// TwinCAT 3 PLC project OnGantryRTC_PLC
// ProgramVersion: 3.1.4020.4
// libraries:
//   Tc2_EtherCAT, * (Beckhoff Automation GmbH)
//   Tc2_Standard, * (Beckhoff Automation GmbH)
//   Tc2_System, * (Beckhoff Automation GmbH)
//   Tc3_Module, * (Beckhoff Automation GmbH)
// project tree:
//   / PlcTask.TcTTO
//   POUs/ BeamEnChain.TcPOU, bsm.TcPOU, Ehercat_Manage.TcPOU, F_scale_int_real.TcPOU, F_scale_real_int.TcPOU, OnGantry_IO.TcPOU
// real-time tasks:
//   TASK Task10ms: cycle T#10ms, priority 10, ADS port 350
//   TASK Task5ms: cycle T#5ms, priority 1, ADS port 351
//   TASK PlcTask: cycle T#10ms, priority 20, ADS port 352
// I/O:
//   DEVICE PCI, AmsNetId 192.168.60.2.2.1
//     Term 1 (EK1200) [EK1200-5000 EtherCAT Power supply (2A E-Bus)]
//       Term 2 (EL1809) [EL1809 16Ch. Dig. Input 24V, 3ms]
//       Term 3 (EL2809) [EL2809 16Ch. Dig. Output 24V, 0.5A]
//       Term 4 (EL6751) [EL6751 CANopen Master]
//       Term 5 (EL9011) [EL9011 End Terminal]
//   DEVICE MasterOut, AmsNetId 192.168.60.2.7.1
//     SlaveBSM [CX2030 EtherCAT slave]
//     SlaveBGM [CX2030 EtherCAT slave]
//     SlaveIGS [CX2030 EtherCAT slave]
//   DEVICE MasterIn (disabled), AmsNetId 192.168.60.2.4.1
//   DEVICE Device 5 (USB)
//     Box 1 (CX2100 Power Supply)
//     Box 254 (C9900-L100 License-Key-USB-Stick)
//   DEVICE CANOpenMaster, AmsNetId 192.168.60.2.3.1
//     Box 1 (EL6751)
//   DEVICE NRT
// variable links:
//   CANOpenMaster <-> RTC_StateMachine/ThreadFSM
//     Box 1 (EL6751)/Inputs/NodeState <-> FmDevices/CANOpen
//     Box 1 (EL6751)/RxPDO 1/Outputs/CurrentState <-> OutputsOGR/CurrentState
//     Box 1 (EL6751)/RxPDO 1/Outputs/DoseSegment <-> OutputsOGR/DoseSegment
//     Box 1 (EL6751)/RxPDO 1/Outputs/DoseTotal <-> OutputsOGR/DoseTotal
//     Box 1 (EL6751)/RxPDO 1/Outputs/IUT <-> OutputsOGR/IUT
//     Box 1 (EL6751)/RxPDO 2/Outputs/CollimatorDegree <-> OutputsBsm/CollimatorDegree
//     Box 1 (EL6751)/TxPDO 1/Inputs/CurrentState <-> InputsOGR/CurrentState
//     Box 1 (EL6751)/TxPDO 1/Inputs/GantryAngle <-> InputsOGR/GantryAngle
//     Box 1 (EL6751)/TxPDO 1/Inputs/GantrySpeed <-> InputsOGR/GantrySpeed
//     Box 1 (EL6751)/TxPDO 1/Inputs/IUT <-> InputsOGR/IUT
//     Box 1 (EL6751)/TxPDO 1/Inputs/RadiationIndex <-> InputsOGR/RadiationIndex
//     Box 1 (EL6751)/TxPDO 2/Inputs/FieldDefiningLamp <-> InputsBsm/FieldLightFrmBSC
//     Box 1 (EL6751)/TxPDO 2/Inputs/FkpButton <-> InputsOGR/FkpButton
//     Box 1 (EL6751)/TxPDO 2/Inputs/OdiLight <-> InputsBsm/OdiLight
//     Box 1 (EL6751)/TxPDO 3/Inputs/BsmMotionEnable <-> InputsBsm/BsmMotionEnable
//     Box 1 (EL6751)/TxPDO 3/Inputs/HHCWheel1 <-> InputsBsm/WheelBsm1
//     Box 1 (EL6751)/TxPDO 3/Inputs/HHCWheel2 <-> InputsBsm/WheelBsm2
//     Box 1 (EL6751)/TxPDO 3/Inputs/HHCWheel3 <-> InputsBsm/WheelBsm3
//   MasterOut <-> RTC_StateMachine/ThreadFSM
//     SlaveBGM/IO Inputs/BankIndex <-> InputsBgmPlan/BankIndex
//     SlaveBGM/IO Inputs/BeamID <-> InputsBgmPlan/BeamID
//     SlaveBGM/IO Inputs/CPIndex <-> InputsBgmPlan/CPIndex
//     SlaveBGM/IO Inputs/CPTotal <-> InputsBgmPlan/CPTotal
//     SlaveBGM/IO Inputs/Crc32 <-> InputsBgmPlan/Crc32
//     SlaveBGM/IO Inputs/DoseSegment <-> InputsDose/DoseSegment
//     SlaveBGM/IO Inputs/DoseTotal <-> InputsDose/DoseTotal
//     SlaveBGM/IO Inputs/RadiationIndex <-> InputsBeam/RadiationIndex
//     SlaveBGM/IO Inputs/WatchDogOk <-> FmDevices/BgmWdOk
//     SlaveBGM/IO Inputs/bgm_interlocks <-> InputsSubFsm/BgmInterlocks
//     SlaveBGM/IO Inputs/bgm_last_state <-> InputsSubFsm/BgmLastState
//     SlaveBGM/IO Inputs/bgm_required_state <-> InputsSubFsm/BgmRequiredState
//     SlaveBGM/IO Inputs/bgm_state <-> InputsSubFsm/BgmCurrentState
//     SlaveBGM/IO Inputs/bgm_unready1 <-> InputsSubFsm/BgmUnreadys
//     SlaveBGM/IO Outputs/BankIndex <-> OutputsBgmPlan/BankIndex
//     SlaveBGM/IO Outputs/BeamID <-> OutputsBgmPlan/BeamID
//     SlaveBGM/IO Outputs/CPIndex <-> OutputsBgmPlan/CPIndex
//     SlaveBGM/IO Outputs/CPTotal <-> OutputsBgmPlan/CPTotal
//     SlaveBGM/IO Outputs/Crc32 <-> OutputsBgmPlan/Crc32
//     SlaveBGM/IO Outputs/DoseInterlockEnable <-> OutputsDose/DoseInterlockEnable
//     SlaveBGM/IO Outputs/DoseTotal <-> OutputsBgmPlan/DoseTotal
//     SlaveBGM/IO Outputs/PlanData <-> OutputsBgmPlan/Data
//     SlaveBGM/IO Outputs/QuickBeamTotalSet1 <-> OutputsBeam/beam_total_set1
//     SlaveBGM/IO Outputs/RadiationIndex <-> OutputsOGR/RadiationIndex
//     SlaveBGM/IO Outputs/RequiredState <-> OutputsSubFsm/BgmRequiredState
//     SlaveBGM/IO Outputs/ServoAxisType <-> OutputsBgmPlan/ServoAxisType
//     SlaveBGM/InfoData/State <-> FmDevices/BGMSlave
//     SlaveBSM/IO Inputs/BankIndex <-> InputsBsm/BankIndex
//     SlaveBSM/IO Inputs/BeamId <-> InputsBsm/BeamID
//     SlaveBSM/IO Inputs/BsmReady <-> InputsBsm/BsmReady
//     SlaveBSM/IO Inputs/CollimatorPosition <-> InputsBsm/CollimatorPosition
//     SlaveBSM/IO Inputs/CpIndex <-> InputsBsm/CPIndex
//     SlaveBSM/IO Inputs/CpTotal <-> InputsBsm/CPTotal
//     SlaveBSM/IO Inputs/Crc32 <-> InputsBsm/Crc32
//     SlaveBSM/IO Inputs/CurrentState <-> InputsBsm/CurrentState
//     SlaveBSM/IO Inputs/Data <-> InputsBsm/PosFeedback
//     SlaveBSM/IO Inputs/HeadP1 <-> InputsBsm/HeadP1
//     SlaveBSM/IO Inputs/HeaddSpeed <-> InputsBsm/HeadSpeed
//     SlaveBSM/IO Inputs/Headp2 <-> InputsBsm/HeadP2
//     SlaveBSM/IO Inputs/InitModeAck <-> InputsBsm/BSMInitModeAck
//     SlaveBSM/IO Inputs/InitResult1 <-> InputsBsm/InitResult1
//     SlaveBSM/IO Inputs/InitResult2 <-> InputsBsm/InitResult2
//     SlaveBSM/IO Inputs/Interlock <-> InputsBsm/Interlock
//     SlaveBSM/IO Inputs/JawMaxSpeed <-> InputsBsm/JawMaxSpeed
//     SlaveBSM/IO Inputs/LastState <-> InputsBsm/LastState
//     SlaveBSM/IO Inputs/LeafMaxSpeed <-> InputsBsm/LeafMaxSpeed
//     SlaveBSM/IO Inputs/RadiationIndex <-> InputsBsm/RadiationIndex
//     SlaveBSM/IO Inputs/Status <-> InputsBsm/Status
//     SlaveBSM/IO Inputs/UpJaw1P1 <-> InputsBsm/UpJaw1P1
//     SlaveBSM/IO Inputs/UpJaw1P2 <-> InputsBsm/UpJaw1P2
//     SlaveBSM/IO Inputs/UpJaw2P1 <-> InputsBsm/UpJaw2P1
//     SlaveBSM/IO Inputs/UpJaw2P2 <-> InputsBsm/UpJaw2P2
//     SlaveBSM/IO Outputs/BSMInitMode <-> OutputsBsm/BSMInitMode
//     SlaveBSM/IO Outputs/BSMOK <-> OutputsBsm/BsmOk
//     SlaveBSM/IO Outputs/BankIndex <-> OutputsBsm/BankIndex
//     SlaveBSM/IO Outputs/BeamId <-> OutputsBsm/BeamID
//     SlaveBSM/IO Outputs/CalibrationJaw <-> OutputsBsm/CalibrationJaw
//     SlaveBSM/IO Outputs/CollimatorPosition <-> OutputsBsm/CollimatorPosition
//     SlaveBSM/IO Outputs/Commands <-> OutputsBsm/Commands
//     SlaveBSM/IO Outputs/CpIndex <-> OutputsBsm/CPIndex
//     SlaveBSM/IO Outputs/CpTotal <-> OutputsBsm/CPTotal
//     SlaveBSM/IO Outputs/Crc32 <-> OutputsBsm/Crc32
//     SlaveBSM/IO Outputs/Data <-> OutputsBsm/Data
//     SlaveBSM/IO Outputs/HHCFunctionCode <-> OutputsBsm/HhcFunctionCode
//     SlaveBSM/IO Outputs/HHCVoltage <-> OutputsBsm/HhcVoltage
//     SlaveBSM/IO Outputs/HHCWheel1 <-> OutputsBsm/HHCWheel1
//     SlaveBSM/IO Outputs/HHCWheel2 <-> OutputsBsm/HHCWheel2
//     SlaveBSM/IO Outputs/HHCWheel3 <-> OutputsBsm/HHCWheel3
//     SlaveBSM/IO Outputs/HeadAngle <-> OutputsBsm/HeadAngle
//     SlaveBSM/IO Outputs/HeadAngleK <-> OutputsBsm/HeadAngleK
//     SlaveBSM/IO Outputs/HeadAngleOffset <-> OutputsBsm/HeadAngleOffset
//     SlaveBSM/IO Outputs/HeadAngleSecondaryK <-> OutputsBsm/HeadAngleSecondaryK
//     SlaveBSM/IO Outputs/HeadLimitEncoder <-> OutputsBsm/HeadLimitEncoder
//     SlaveBSM/IO Outputs/HeadSpeed <-> OutputsBsm/HeadSpeed
//     SlaveBSM/IO Outputs/HeadTolerance <-> OutputsBsm/HeadTolerance
//     SlaveBSM/IO Outputs/HwEnable <-> OutputsBsm/HwEnable
//     SlaveBSM/IO Outputs/JawXTolerance <-> OutputsBsm/ToleranceJawX
//     SlaveBSM/IO Outputs/JawYTolerance <-> OutputsBsm/ToleranceJawY
//     SlaveBSM/IO Outputs/LeafTolerance <-> OutputsBsm/ToleranceLeaf
//     SlaveBSM/IO Outputs/RadiationIndex <-> OutputsBsm/RadiationIndex
//     SlaveBSM/IO Outputs/RequiredState <-> OutputsBsm/RequiredState
//     SlaveBSM/IO Outputs/UpJaw1Pos <-> OutputsBsm/UpJaw1Pos
//     SlaveBSM/IO Outputs/UpJaw2Pos <-> OutputsBsm/UpJaw2Pos
//     SlaveBSM/IO Outputs/UpJaw1Speed <-> OutputsBsm/UpJaw1Speed
//     SlaveBSM/IO Outputs/UpJaw2Speed <-> OutputsBsm/UpJaw2Speed
//     SlaveBSM/InfoData/State <-> FmDevices/BSMSlave
//     SlaveIGS/IO Inputs/CollimatorCross <-> InputsIgsSlv/CollimatorCross
//     SlaveIGS/IO Inputs/CollimatorLong <-> InputsIgsSlv/CollimatorLong
//     SlaveIGS/IO Inputs/CollimatorOffsetCross <-> InputsIgsSlv/CollimatorOffsetCross
//     SlaveIGS/IO Inputs/CollimatorOffsetLong <-> InputsIgsSlv/CollimatorOffsetLong
//     SlaveIGS/IO Inputs/CollimatorPosReady <-> InputsIgsSlv/CollimatorPosReady
//     SlaveIGS/IO Inputs/CurrentState <-> InputsIgsSlv/CurrentState
//     SlaveIGS/IO Inputs/HighVoltageGeneratorErrorCode <-> InputsIgsSlv/HighVoltageGeneratorErrorCode
//     SlaveIGS/IO Inputs/ICUFocusExpActual <-> InputsIgsSlv/IcuFocusExpActual
//     SlaveIGS/IO Inputs/ICUFrequencyExpActual <-> InputsIgsSlv/IcuFrequencyExpActual
//     SlaveIGS/IO Inputs/ICUKVExpActual <-> InputsIgsSlv/IcuKVExpActual
//     SlaveIGS/IO Inputs/ICUMAExpActual <-> InputsIgsSlv/IcuMAExpActual
//     SlaveIGS/IO Inputs/ICUMSExpActual <-> InputsIgsSlv/IcuMSExpActual
//     SlaveIGS/IO Inputs/IcuErrorCode <-> InputsIgsSlv/IcuErrorCode
//     SlaveIGS/IO Inputs/Interlock <-> InputsIgsSlv/Interlock
//     SlaveIGS/IO Inputs/KVEncode1 <-> InputsIgsSlv/KVEncode1
//     SlaveIGS/IO Inputs/KVEncode2 <-> InputsIgsSlv/KVEncode2
//     SlaveIGS/IO Inputs/KVPosActual <-> InputsIgsSlv/KVPosActual
//     SlaveIGS/IO Inputs/KVPosReady <-> InputsIgsSlv/KVPosReady
//     SlaveIGS/IO Inputs/KvPanelErrorcode <-> InputsIgsSlv/KvPanelErrorcode
//     SlaveIGS/IO Inputs/LastState <-> InputsIgsSlv/LastState
//     SlaveIGS/IO Inputs/MVEncode1 <-> InputsIgsSlv/MVEncode1
//     SlaveIGS/IO Inputs/MVEncode2 <-> InputsIgsSlv/MVEncode2
//     SlaveIGS/IO Inputs/MVPanelErrorcode <-> InputsIgsSlv/MVPanelErrorcode
//     SlaveIGS/IO Inputs/MVPosActual <-> InputsIgsSlv/MVPosActual
//     SlaveIGS/IO Inputs/MVPosReady <-> InputsIgsSlv/MVPosReady
//     SlaveIGS/IO Inputs/RecordCounter <-> InputsIgsSlv/RecordCounter
//     SlaveIGS/IO Inputs/RecordFlag <-> InputsIgsSlv/RecordFlag
//     SlaveIGS/IO Inputs/WatchDogOk <-> FmDevices/IgsWdOk
//     SlaveIGS/IO Outputs/CollimatorCross <-> OutputsIgsSlv/CollimatorCross
//     SlaveIGS/IO Outputs/CollimatorLong <-> OutputsIgsSlv/CollimatorLong
//     SlaveIGS/IO Outputs/CollimatorOffsetCross <-> OutputsIgsSlv/CollimatorOffsetCross
//     SlaveIGS/IO Outputs/CollimatorOffsetLong <-> OutputsIgsSlv/CollimatorOffsetLong
//     SlaveIGS/IO Outputs/ICUFocusExp <-> OutputsIgsSlv/IcuFocusExp
//     SlaveIGS/IO Outputs/ICUFrequencyExp <-> OutputsIgsSlv/IcuFrequencyExp
//     SlaveIGS/IO Outputs/ICUKVExp <-> OutputsIgsSlv/IcuKVExp
//     SlaveIGS/IO Outputs/ICUMAExp <-> OutputsIgsSlv/IcuMAExp
//     SlaveIGS/IO Outputs/ICUMSExp <-> OutputsIgsSlv/IcuMSExp
//     SlaveIGS/IO Outputs/KVOffset1 <-> OutputsIgsSlv/KVOffset1
//     SlaveIGS/IO Outputs/KVOffset2 <-> OutputsIgsSlv/KVOffset2
//     SlaveIGS/IO Outputs/KVPosTarget <-> OutputsIgsSlv/KVPosTarget
//     SlaveIGS/IO Outputs/KvTimeout <-> OutputsIgsSlv/KvTimeout
//     SlaveIGS/IO Outputs/MVOffset1 <-> OutputsIgsSlv/MVOffset1
//     SlaveIGS/IO Outputs/MVOffset2 <-> OutputsIgsSlv/MVOffset2
//     SlaveIGS/IO Outputs/MVPosTarget <-> OutputsIgsSlv/MVPosTarget
//     SlaveIGS/IO Outputs/MvTimeout <-> OutputsIgsSlv/MvTimeout
//     SlaveIGS/IO Outputs/PlanTotalFrame <-> OutputsIgsSlv/PlanTotalFrame
//     SlaveIGS/IO Outputs/RequiredState <-> OutputsIgsSlv/RequiredState
//     SlaveIGS/IO Outputs/Reset <-> OutputsIgsSlv/Reset
//     SlaveIGS/IO Outputs/WorkMode <-> OutputsIgsSlv/WorkMode
//     SlaveIGS/InfoData/State <-> FmDevices/IGSSlave
//   MasterOut <-> TCPServer/ThreadGUI
//     SlaveBGM/IO Inputs/BgmHalEmulate <-> InputsHalState/EmulateState/BGM
//     SlaveBGM/IO Inputs/DoseDelta <-> InputsBeam/DoseDelta
//     SlaveBGM/IO Inputs/DoseInformation1 <-> InputsDose/DoseInformation1
//     SlaveBGM/IO Inputs/DoseInformation2 <-> InputsDose/DoseInformation2
//     SlaveBGM/IO Inputs/GunCathodCurrentRead <-> InputsGun/gun_cathode_current_read
//     SlaveBGM/IO Inputs/GunFilaCurrentRead <-> InputsGun/gun_fila_current_read
//     SlaveBGM/IO Inputs/GunFilaVolRead <-> InputsGun/gun_fila_vol_read
//     SlaveBGM/IO Inputs/GunHvRead <-> InputsGun/gun_hv_read
//     SlaveBGM/IO Inputs/GunRemainingTime <-> InputsGun/GunRemainingTime
//     SlaveBGM/IO Inputs/afc_RF_AI <-> InputsAfc/afc_RF_AI
//     SlaveBGM/IO Inputs/afc_current_pos <-> InputsAfc/afc_current_pos
//     SlaveBGM/IO Inputs/afc_mode <-> InputsAfc/afc_mode
//     SlaveBGM/IO Inputs/beam_dose_rate_read1 <-> InputsBeam/beam_dose_rate_read1
//     SlaveBGM/IO Inputs/beam_dose_rate_read2 <-> InputsBeam/beam_dose_rate_read2
//     SlaveBGM/IO Inputs/beam_total_read1 <-> InputsBeam/beam_total_read1
//     SlaveBGM/IO Inputs/beam_total_read2 <-> InputsBeam/beam_total_read2
//     SlaveBGM/IO Inputs/mod_app_ver <-> InputsModulator/mod_app_ver
//     SlaveBGM/IO Inputs/mod_average_power_read <-> InputsModulator/mod_average_power_read
//     SlaveBGM/IO Inputs/mod_dc_vol_read <-> InputsModulator/mod_dc_vol_read
//     SlaveBGM/IO Inputs/mod_dc_voltage_rb <-> InputsModulator/mod_dc_voltage_set_read
//     SlaveBGM/IO Inputs/mod_filament_current_read <-> InputsModulator/mod_filament_current_read
//     SlaveBGM/IO Inputs/mod_filament_vol_rb <-> InputsModulator/mod_filament_vol_set_read
//     SlaveBGM/IO Inputs/mod_filament_vol_read <-> InputsModulator/mod_filament_vol_read
//     SlaveBGM/IO Inputs/mod_fpga_ver <-> InputsModulator/mod_fpga_ver
//     SlaveBGM/IO Inputs/mod_hv_hour <-> InputsModulator/mod_hv_hour
//     SlaveBGM/IO Inputs/mod_hv_interlock <-> InputsModulator/mod_hv_interlock
//     SlaveBGM/IO Inputs/mod_level <-> InputsModulator/mod_level
//     SlaveBGM/IO Inputs/mod_off_hour <-> InputsModulator/mod_off_hour
//     SlaveBGM/IO Inputs/mod_pluse_width_rb <-> InputsModulator/mod_pulse_width_set_read
//     SlaveBGM/IO Inputs/mod_prf_read <-> InputsModulator/mod_prf_read
//     SlaveBGM/IO Inputs/mod_pulse_width_read <-> InputsModulator/mod_pulse_width_read
//     SlaveBGM/IO Inputs/mod_remaining_time <-> InputsModulator/mod_remaining_time
//     SlaveBGM/IO Inputs/mod_standby_hour <-> InputsModulator/mod_standby_hour
//     SlaveBGM/IO Inputs/mod_standby_interlock <-> InputsModulator/mod_standby_interlock
//     SlaveBGM/IO Inputs/mod_state_rb <-> InputsModulator/mod_state_set_read
//     SlaveBGM/IO Inputs/mod_state_read <-> InputsModulator/mod_state_read
//     SlaveBGM/IO Inputs/mod_trig_hour <-> InputsModulator/mod_trig_hour
//     SlaveBGM/IO Inputs/mod_trig_interlock <-> InputsModulator/mod_trig_interlock
//     SlaveBGM/IO Inputs/sf6_pressure <-> InputsSF6/sf6_pressure
//     SlaveBGM/IO Inputs/vac_current <-> InputsVac/vac_current
//     SlaveBGM/IO Inputs/vac_voltage <-> InputsVac/vac_voltage
//     SlaveBGM/IO Inputs/water_flow_in <-> InputsWater/water_flow_in
//     SlaveBGM/IO Inputs/water_flow_low_set <-> InputsWater/water_flow_low_set
//     SlaveBGM/IO Inputs/water_flow_switch <-> InputsWater/water_flow_switch
//     SlaveBGM/IO Inputs/water_interlock_raw <-> InputsWater/water_interlock_raw
//     SlaveBGM/IO Inputs/water_pressure_in <-> InputsWater/water_pressure
//     SlaveBGM/IO Inputs/water_temp_{1..5} <-> InputsWater/water_temp_{1..5}  (5 links)
//     SlaveBGM/IO Inputs/water_temp_back <-> InputsWater/water_temp_back
//     SlaveBGM/IO Inputs/water_temp_high_set <-> InputsWater/water_temp_high_set
//     SlaveBGM/IO Inputs/water_temp_in <-> InputsWater/water_temp_in
//     SlaveBGM/IO Inputs/water_temp_low_set <-> InputsWater/water_temp_low_set
//     SlaveBGM/IO Outputs/AfcRfSet <-> OutputsAfc/afc_RF_set
//     SlaveBGM/IO Outputs/DPP <-> OutputsPrf/DPP
//     SlaveBGM/IO Outputs/DarkCurrentLimit <-> OutputsDose/DarkCurrentLimit
//     SlaveBGM/IO Outputs/DoseCalFactorA1 <-> OutputsDose/DoseCalFactorA1
//     SlaveBGM/IO Outputs/DoseCalFactorA2 <-> OutputsDose/DoseCalFactorA2
//     SlaveBGM/IO Outputs/DoseCalFactorB1 <-> OutputsDose/DoseCalFactorB1
//     SlaveBGM/IO Outputs/DoseCalFactorB2 <-> OutputsDose/DoseCalFactorB2
//     SlaveBGM/IO Outputs/DoseDeltaActionRange <-> OutputsPrf/DoseDeltaActionRange
//     SlaveBGM/IO Outputs/DoseOverrangeRatio <-> OutputsDose/SegmentOverrangeRatio
//     SlaveBGM/IO Outputs/DoseRateAccTime <-> OutputsDose/DoseRateAccTime
//     SlaveBGM/IO Outputs/DoseRateCycleTime <-> OutputsDose/DoseRateCycleTime
//     SlaveBGM/IO Outputs/DoseRateLimit <-> OutputsDose/DoseRateLimit
//     SlaveBGM/IO Outputs/DualChannelRatio <-> OutputsDose/DualChannelRatio
//     SlaveBGM/IO Outputs/DualChannelTolerance <-> OutputsDose/DualChannelTolerance
//     SlaveBGM/IO Outputs/DummyDoseRateSet <-> OutputsDose/DummyDoseRateSet
//     SlaveBGM/IO Outputs/PrfCatchCurveD1 <-> OutputsPrf/PrfCatchCurveD1
//     SlaveBGM/IO Outputs/PrfCatchCurveD2 <-> OutputsPrf/PrfCatchCurveD2
//     SlaveBGM/IO Outputs/PrfCatchCurveP1 <-> OutputsPrf/PrfCatchCurveP1
//     SlaveBGM/IO Outputs/PrfCatchCurveP2 <-> OutputsPrf/PrfCatchCurveP2
//     SlaveBGM/IO Outputs/PrfCatchCurveQ1 <-> OutputsPrf/PrfCatchCurveQ1
//     SlaveBGM/IO Outputs/PrfCatchCurveQ2 <-> OutputsPrf/PrfCatchCurveQ2
//     SlaveBGM/IO Outputs/PrfCatchCurveR1 <-> OutputsPrf/PrfCatchCurveR1
//     SlaveBGM/IO Outputs/PrfCatchCurveR2 <-> OutputsPrf/PrfCatchCurveR2
//     SlaveBGM/IO Outputs/PrfCatchCycle <-> OutputsPrf/PrfCatchCycle
//     SlaveBGM/IO Outputs/PrfDeltaRatio <-> OutputsPrf/PrfDeltaRatio
//     SlaveBGM/IO Outputs/PrfRatio <-> OutputsPrf/PrfRatio
//     SlaveBGM/IO Outputs/QuickBeamProtectTimeSet <-> OutputsBeam/beam_time_set
//     SlaveBGM/IO Outputs/QuickBeamTotalSet2 <-> OutputsBeam/beam_total_set2
//     SlaveBGM/IO Outputs/SymmetryThreshold1 <-> OutputsDose/SymmetryThreshold1
//     SlaveBGM/IO Outputs/SymmetryThreshold2 <-> OutputsDose/SymmetryThreshold2
//     SlaveBGM/IO Outputs/SymmetryTolerance1 <-> OutputsDose/SymmetryTolerance1
//     SlaveBGM/IO Outputs/SymmetryTolerance2 <-> OutputsDose/SymmetryTolerance2
//     SlaveBGM/IO Outputs/afc_dir_swap <-> OutputsAfc/afc_dir_swap
//     SlaveBGM/IO Outputs/afc_linear_high <-> OutputsAfc/afc_linear_high
//     SlaveBGM/IO Outputs/afc_linear_low <-> OutputsAfc/afc_linear_low
//     SlaveBGM/IO Outputs/afc_manual_dir <-> OutputsAfc/afc_manual_dir
//     SlaveBGM/IO Outputs/afc_manual_move <-> OutputsAfc/afc_manual_move
//     SlaveBGM/IO Outputs/afc_mode_set <-> OutputsAfc/afc_mode_set
//     SlaveBGM/IO Outputs/afc_motor_max_speed <-> OutputsAfc/afc_motor_max_speed
//     SlaveBGM/IO Outputs/afc_preset <-> OutputsAfc/afc_preset
//     SlaveBGM/IO Outputs/emulator_enable <-> OutputsHalState/BgmEmulate
//     SlaveBGM/IO Outputs/gui_cmd_reset <-> OutputsFsm/reset_command
//     SlaveBGM/IO Outputs/gun_cathode_current_max <-> OutputsGun/gun_cathode_current_max
//     SlaveBGM/IO Outputs/gun_cathode_current_min <-> OutputsGun/gun_cathode_current_min
//     SlaveBGM/IO Outputs/gun_cathode_current_rat_2 <-> OutputsGun/gun_cathode_current_rat_2
//     SlaveBGM/IO Outputs/gun_dr_at_fullpower <-> OutputsGun/gun_dr_at_fullpower
//     SlaveBGM/IO Outputs/gun_fila_current_rat_2 <-> OutputsGun/gun_fila_current_rat_2
//     SlaveBGM/IO Outputs/gun_fila_current_set_tol <-> OutputsGun/gun_fila_current_set_tol
//     SlaveBGM/IO Outputs/gun_fila_vol_max <-> OutputsGun/gun_fila_vol_max
//     SlaveBGM/IO Outputs/gun_fila_vol_min <-> OutputsGun/gun_fila_vol_min
//     SlaveBGM/IO Outputs/gun_fila_vol_rat_2 <-> OutputsGun/gun_fila_vol_rat_2
//     SlaveBGM/IO Outputs/gun_fila_vol_set_rat_{1..4} <-> OutputsGun/gun_fila_vol_set_rat_{1..4}  (4 links)
//     SlaveBGM/IO Outputs/gun_heaterok_judgetime <-> OutputsGun/gun_heaterok_judgetime
//     SlaveBGM/IO Outputs/gun_hv <-> OutputsGun/gun_hv
//     SlaveBGM/IO Outputs/gun_hv_rat_{1..4} <-> OutputsGun/gun_hv_rat_{1..4}  (4 links)
//     SlaveBGM/IO Outputs/gun_hv_read_rat2 <-> OutputsGun/gun_hv_read_rat2
//     SlaveBGM/IO Outputs/gun_rundown_dr_k <-> OutputsGun/gun_rundown_dr_k
//     SlaveBGM/IO Outputs/gun_rundown_prf_k <-> OutputsGun/gun_rundown_prf_k
//     SlaveBGM/IO Outputs/gun_warmup <-> OutputsGun/gun_warmup
//     SlaveBGM/IO Outputs/gun_warmup_time <-> OutputsGun/gun_warmup_time
//     SlaveBGM/IO Outputs/mod_dc_voltage <-> OutputsModulator/mod_dc_voltage
//     SlaveBGM/IO Outputs/mod_filament_vol <-> OutputsModulator/mod_filament_vol
//     SlaveBGM/IO Outputs/mod_pulse_width <-> OutputsModulator/mod_pluse_width
//     SlaveBGM/IO Outputs/prf_set <-> OutputsPrf/prf_set
//     SlaveIGS/IO Inputs/HVGeneratorHU <-> InputsIgs/HVGeneratorHU
//     SlaveIGS/IO Outputs/KvTorlerance <-> OutputsIgs/KvTorlerance
//     SlaveIGS/IO Outputs/MvTorlerance <-> OutputsIgs/MvTorlerance
//   OnGantryRTC_PLC/OnGantryRTC_PLC Instance <-> MasterOut
//     PlcTask Inputs/Ehercat_Manage.arrbyNetId <-> InfoData/AmsNetId
//   OnGantryRTC_PLC/OnGantryRTC_PLC Instance <-> PCI/Term 1 (EK1200)/Term 2 (EL1809)
//     PlcTask Inputs/OnGantry_IO.plc_to_io_OnGantryRtcWdOK <-> Channel 3/Input
//     PlcTask Inputs/OnGantry_IO.plc_to_io_bAutoMove <-> Channel 2/Input
//     PlcTask Inputs/OnGantry_IO.plc_to_io_bGantryTouchGuard <-> Channel 1/Input
//   OnGantryRTC_PLC/OnGantryRTC_PLC Instance <-> PCI/Term 1 (EK1200)/Term 3 (EL2809)
//     PlcTask Outputs/OnGantry_IO.plc_to_io_OnGantryMoveEn <-> Channel 3/Output
//     PlcTask Outputs/OnGantry_IO.plc_to_io_bCanOpenOk <-> Channel 1/Output
//     PlcTask Outputs/OnGantry_IO.plc_to_io_bEthercatInOk <-> Channel 2/Output
//     PlcTask Outputs/OnGantry_IO.plc_to_io_bEthercatOutOk <-> Channel 4/Output
//     PlcTask Outputs/OnGantry_IO.plc_to_io_bKvEn <-> Channel 7/Output
//     PlcTask Outputs/OnGantry_IO.plc_to_io_bSwManualMotionEn <-> Channel 9/Output
//     PlcTask Outputs/OnGantry_IO.plc_to_io_bSwRest <-> Channel 6/Output
//     PlcTask Outputs/OnGantry_IO.plc_to_io_bSwWatchDogService <-> Channel 5/Output
//   OnGantryRTC_PLC/OnGantryRTC_PLC Instance <-> RTC_StateMachine/ThreadFSM
//     PlcTask Inputs/OnGantry_IO.plc_to_cpp_OnGantryMoveEn <-> OutputsOnGantryHD/SwOnGantryMoveEn
//     PlcTask Inputs/OnGantry_IO.plc_to_cpp_bCanOpenOk <-> OutputsOnGantryHD/SwCanOpenOk
//     PlcTask Inputs/OnGantry_IO.plc_to_cpp_bEthercatInOk <-> OutputsOnGantryHD/SwEthercatInOk
//     PlcTask Inputs/OnGantry_IO.plc_to_cpp_bEthercatOutOk <-> OutputsOnGantryHD/SwEthercatOutOk
//     PlcTask Inputs/OnGantry_IO.plc_to_cpp_bKvEn <-> OutputsOnGantryHD/SwKvEn
//     PlcTask Inputs/OnGantry_IO.plc_to_cpp_bSwManualMotionEn <-> OutputsFsm/bSwManualMotionEn
//     PlcTask Outputs/OnGantry_IO.plc_to_cpp_OnGantryRtcWdOK <-> FmDevices/OnGantryRTCWdOk
//     PlcTask Outputs/OnGantry_IO.plc_to_cpp_bAutoMove <-> InputsOnGantryHD/AutoMoveEn
//     PlcTask Outputs/OnGantry_IO.plc_to_cpp_bGantryTouchGuard <-> InputsOnGantryHD/GantryTouchGuard
//   OnGantryRTC_PLC/OnGantryRTC_PLC Instance <-> TCPServer/ThreadGUI
//     PlcTask Inputs/Ehercat_Manage.bResetState <-> OutputsFsm/reset_command
//     PlcTask Inputs/OnGantry_IO.plc_to_cpp_bSwRest <-> OutputsFsm/reset_command
//   RTC_StateMachine/ThreadFSM <-> TCPServer/ThreadGUI
//     InputsBeam/DoseRateSet <-> OutputsBeam/beam_dose_rate_set
//     InputsBeam/beam_total_set1 <-> OutputsBeam/beam_total_set1
//     InputsBsmFmGUI/BSMEnalbe <-> OutputsBsm/BSMEnable
//     InputsBsmFmGUI/BSMInitMode <-> OutputsBsm/BSMInitMode
//     InputsBsmFmGUI/BSMOk <-> OutputsBsm/bsm_ok
//     InputsBsmFmGUI/CalibrationJaw <-> OutputsBsm/CalibrationJaw
//     InputsBsmFmGUI/CollimatorPosition <-> OutputsBsm/CollimatorPosition
//     InputsBsmFmGUI/EmulatorEnable <-> OutputsHalState/BsmEmulate
//     InputsBsmFmGUI/HeadAnagle <-> OutputsBsm/HeadAngle
//     InputsBsmFmGUI/HeadAngleK <-> OutputsBsm/HeadAngleK
//     InputsBsmFmGUI/HeadAngleOffset <-> OutputsBsm/HeadAngleOffset
//     InputsBsmFmGUI/HeadAngleSecondaryK <-> OutputsBsm/HeadAngleSecondaryK
//     InputsBsmFmGUI/HeadLimitEncoder <-> OutputsBsm/HeadLimitEncoder
//     InputsBsmFmGUI/HeadSpeed <-> OutputsBsm/bsm_Head_speed
//     InputsBsmFmGUI/UpJaw1Speed <-> OutputsBsm/bsm_up_jaw1_speed
//     InputsBsmFmGUI/UpJaw2Speed <-> OutputsBsm/bsm_up_jaw2_speed
//     InputsCtrlState/ControllerEmuMode <-> OutputsHalState/ControllerEmuSet
//     InputsDose/DoseInterlockEnable <-> OutputsDose/DoseInterlockEnable
//     InputsFsm/ParaCrcStatus <-> OutputsFsm/ParaCrcStatus
//     InputsFsm/com_status_gui <-> OutputsFsm/ComStateGUI
//     InputsFsm/gui_cmd{1..8} <-> OutputsFsm/GuiCmd{1..8}  (8 links)
//     InputsIgs/CollimatorCross <-> OutputsIgs/CollimatorCross
//     InputsIgs/CollimatorLong <-> OutputsIgs/CollimatorLong
//     InputsIgs/CollimatorOffsetCross <-> OutputsIgs/CollimatorOffsetCross
//     InputsIgs/CollimatorOffsetLong <-> OutputsIgs/CollimatorOffsetLong
//     InputsIgs/FullHalfShape <-> OutputsIgs/FullHalfShape
//     InputsIgs/IcuFocusExp <-> OutputsIgs/IcuFocusExp
//     InputsIgs/IcuFrequencyExp <-> OutputsIgs/IcuFrequencyExp
//     InputsIgs/IcuKVExp <-> OutputsIgs/IcuKVExp
//     InputsIgs/IcuMAExp <-> OutputsIgs/IcuMAExp
//     InputsIgs/IcuMSExp <-> OutputsIgs/IcuMSExp
//     InputsIgs/KVOffset1 <-> OutputsIgs/KVOffset1
//     InputsIgs/KVOffset2 <-> OutputsIgs/KVOffset2
//     InputsIgs/KVTimeOut <-> OutputsIgs/KVTimeOut
//     InputsIgs/KvWorkPosF <-> OutputsIgs/KvWorkPosF
//     InputsIgs/KvWorkPosH <-> OutputsIgs/KvWorkPosH
//     InputsIgs/MVOffset1 <-> OutputsIgs/MVOffset1
//     InputsIgs/MVOffset2 <-> OutputsIgs/MVOffset2
//     InputsIgs/MVTimeOut <-> OutputsIgs/MVTimeOut
//     InputsIgs/MvWorkPosX <-> OutputsIgs/MvWorkPosX
//     InputsIgs/MvWorkPosY <-> OutputsIgs/MvWorkPosY
//     InputsIgs/Protocal <-> OutputsIgs/Protocal
//     InputsIgs/SynchronousSequence <-> OutputsIgs/SynchronousSequence
//     InputsIgs/WorkMode <-> OutputsIgs/WorkMode
//     InputsVMAT/DoseMaxSpeed <-> OutputsVMAT/DoseMaxSpeed
//     InputsVMAT/GantryMaxSpeed <-> OutputsVMAT/GantryMaxSpeed
//     InputsVMAT/MlcMaxSpeed <-> OutputsVMAT/MlcMaxSpeed
//     OutptsBsmToGUI/BSMStatus <-> InputsBsm/BSMStatus
//     OutptsBsmToGUI/CollimatorPosition <-> InputsBsm/CollimatorPosition
//     OutptsBsmToGUI/EmulatorMode <-> InputsHalState/EmulateState/BSM
//     OutptsBsmToGUI/HeadP1 <-> InputsBsm/bsm_Head_p1
//     OutptsBsmToGUI/HeadP2 <-> InputsBsm/bsm_Head_p2
//     OutptsBsmToGUI/HeadSpeed <-> InputsBsm/HeadSpeed
//     OutptsBsmToGUI/InitResults{0..3} <-> InputsBsm/InitResult{0..3}  (4 links)
//     OutptsBsmToGUI/Jaw1 P1 <-> InputsBsm/bsm_jaw1_p1
//     OutptsBsmToGUI/Jaw1 P2 <-> InputsBsm/bsm_jaw1_p2
//     OutptsBsmToGUI/Jaw2 P1 <-> InputsBsm/bsm_jaw2_p1
//     OutptsBsmToGUI/Jaw2 P2 <-> InputsBsm/bsm_jaw2_p2
//     OutptsBsmToGUI/JawMaxSpeed <-> InputsBsm/JawMaxSpeed
//     OutptsBsmToGUI/LeafMaxSpeed <-> InputsBsm/LeafMaxSpeed
//     OutptsBsmToGUI/MLCActPos <-> InputsBsm/MLCActPos
//     OutputsBeam/RadiationIndex <-> InputsFsm/RadiationIndex
//     OutputsBeam/RadiationTime <-> InputsBeam/beam_time_read
//     OutputsCtrlState/ControllerEmuSet <-> InputsHalState/ControllerEmuMode
//     OutputsCtrlState/WatchDogState <-> InputsHalState/WatchDogState
//     OutputsDose/HighDoseRateInterlock <-> InputsDose/HighDoseRateInterlock
//     OutputsDose/LowDoseRateInterlock <-> InputsDose/LowDoseRateInterlock
//     OutputsFsm/Interlocks <-> InputsFsm/Interlocks
//     OutputsFsm/Terminates <-> InputsFsm/Terminates
//     OutputsFsm/Unreadys <-> InputsFsm/Unreadys
//     OutputsFsm/required_state <-> InputsFsm/RequiredState
//     OutputsFsm/rtc_current_state <-> InputsFsm/CurrentState
//     OutputsFsm/rtc_last_state <-> InputsFsm/LastState
//     OutputsIgs/CollimatorCross <-> InputsIgs/CollimatorCross
//     OutputsIgs/CollimatorLong <-> InputsIgs/CollimatorLong
//     OutputsIgs/CollimatorOffsetCross <-> InputsIgs/CollimatorOffsetCross
//     OutputsIgs/CollimatorOffsetLong <-> InputsIgs/CollimatorOffsetLong
//     OutputsIgs/CollimatorPosReady <-> InputsIgs/CollimatorPosReady
//     OutputsIgs/ExpolistLong <-> InputsIgs/ExposeListLong
//     OutputsIgs/ExposeListGroup <-> InputsIgs/ExposeListGroup
//     OutputsIgs/ExposeListNum <-> InputsIgs/ExposeListNum
//     OutputsIgs/GantryExposeList <-> InputsIgs/ExposeGantryList
//     OutputsIgs/HighVoltageGeneratorErrorCode <-> InputsIgs/HighVoltageGeneratorErrorCode
//     OutputsIgs/IcuErrorCode <-> InputsIgs/IcuErrorCode
//     OutputsIgs/IcuFocusExp <-> InputsIgs/IcuFocusExp
//     OutputsIgs/IcuFrequencyExp <-> InputsIgs/IcuFrequencyExp
//     OutputsIgs/IcuKVExp <-> InputsIgs/IcuKVExp
//     OutputsIgs/IcuMAExp <-> InputsIgs/IcuMAExp
//     OutputsIgs/IcuMSExp <-> InputsIgs/IcuMSExp
//     OutputsIgs/KVOffset1 <-> InputsIgs/KVOffset1
//     OutputsIgs/KVOffset2 <-> InputsIgs/KVOffset2
//     OutputsIgs/KvPanelErrorcode <-> InputsIgs/KvPanelErrorcode
//     OutputsIgs/KvPosReady <-> InputsIgs/KvPosReady
//     OutputsIgs/KvPosition <-> InputsIgs/KvPosition
//     OutputsIgs/MVOffset1 <-> InputsIgs/MVOffset1
//     OutputsIgs/MVOffset2 <-> InputsIgs/MVOffset2
//     OutputsIgs/MVPanelErrorco <-> InputsIgs/MVPanelErrorcode
//     OutputsIgs/MvPosReady <-> InputsIgs/MvPosReady
//     OutputsIgs/MvPosition <-> InputsIgs/MvPosition
//     PlanInputs/BeamEnergyPlan <-> PlanOutputs/BeamEnergyPlan
//     PlanInputs/BeamPlan/AsymxPositionTolerance <-> PlanOutputs/BeamPlan/AsymxPositionTolerance
//     PlanInputs/BeamPlan/AsymyPositionTolerance <-> PlanOutputs/BeamPlan/AsymyPositionTolerance
//     PlanInputs/BeamPlan/BeamLimitingAngleTolerance <-> PlanOutputs/BeamPlan/BeamLimitingAngleTolerance
//     PlanInputs/BeamPlan/BeamNumber <-> PlanOutputs/BeamPlan/BeamNumber
//     PlanInputs/BeamPlan/BeamType <-> PlanOutputs/BeamPlan/BeamType
//     PlanInputs/BeamPlan/Dose <-> PlanOutputs/BeamPlan/Dose
//     PlanInputs/BeamPlan/DoseRateSet <-> PlanOutputs/BeamPlan/DoseRateSet
//     PlanInputs/BeamPlan/GantryAngleTolerance <-> PlanOutputs/BeamPlan/GantryAngleTolerance
//     PlanInputs/BeamPlan/MlcPositionTolerance <-> PlanOutputs/BeamPlan/MlcPositionTolerance
//     PlanInputs/BeamPlan/RadiationType <-> PlanOutputs/BeamPlan/RadiationType
//     PlanInputs/BeamPlan/TableTopLatPositionTolerance <-> PlanOutputs/BeamPlan/TableTopLatPositionTolerance
//     PlanInputs/BeamPlan/TableTopLonPositionTolerance <-> PlanOutputs/BeamPlan/TableTopLonPositionTolerance
//     PlanInputs/BeamPlan/TableTopVerPositionTolerance <-> PlanOutputs/BeamPlan/TableTopVerPositionTolerance
//     PlanInputs/BeamPlan/TotalCP <-> PlanOutputs/BeamPlan/TotalCP
//     PlanInputs/DoseWeight <-> PlanOutputs/DoseWeight
//     PlanInputs/GantryAngle <-> PlanOutputs/GantryAngle
//     PlanInputs/GantryDir <-> PlanOutputs/GantryDir
//     PlanInputs/MlcAngle <-> PlanOutputs/MlcAngle
//     PlanInputs/MlcDir <-> PlanOutputs/MlcDir
//     PlanInputs/MlcPos <-> PlanOutputs/MlcPos
//     PlanInputs/PlanReset <-> PlanOutputs/PlanReset
//     PlanInputs/PssAngle <-> PlanOutputs/PssAngle
//     PlanInputs/PssDir <-> PlanOutputs/PssDir
//     PlanInputs/RecvedCP <-> PlanOutputs/RecvedCP
//     PlanInputs/TableLatPos <-> PlanOutputs/TableLatPos
//     PlanInputs/TableLonPos <-> PlanOutputs/TableLonPos
//     PlanInputs/TablePitchAngle <-> PlanOutputs/TablePitchAngle
//     PlanInputs/TablePitchDir <-> PlanOutputs/TablePitchDir
//     PlanInputs/TableRollAngle <-> PlanOutputs/TableRollAngle
//     PlanInputs/TableRollDir <-> PlanOutputs/TableRollDir
//     PlanInputs/TableVerPos <-> PlanOutputs/TableVerPos
//     PlanOutputs/PlanReady <-> PlanInputs/PlanReady

CONFIGURATION OnGantryRTC_PLC
    RESOURCE PLC ON TwinCAT3
        TASK PlcTask(INTERVAL := T#10ms, PRIORITY := 20);
        PROGRAM Ehercat_Manage WITH PlcTask : Ehercat_Manage;
        PROGRAM bsm WITH PlcTask : bsm;
        PROGRAM BeamEnChain WITH PlcTask : BeamEnChain;
        PROGRAM OnGantry_IO WITH PlcTask : OnGantry_IO;
    END_RESOURCE
END_CONFIGURATION

// ---- POUs/Ehercat_Manage.TcPOU
 PROGRAM Ehercat_Manage
VAR
	(**************************PLC to C++**************************)
	iSlavesCount         AT%Q*          : UINT;	                               //count of slave in device
	wAllState            AT%Q*          : BYTE;                                //bit0:master、bit1:slave1、bit2:slave2...(bit:0=not op 1=op )
	bResetBusy           AT%Q*          : BOOL;                                //0:free ; 1:busy 
	(**************************C++ to PLC**************************)
  	bResetState          AT%I*          : BOOL;                                //activated by a rising edge
	(**************************AMSNETID to T_AmsNetID**************************)
	arrbyNetId           AT%I*          : AMSNETID;                                                                          	
	(**************************Ehercat Manage variables**************************)
	MasterNetId			 		        : T_AmsNetID;//:='192.168.50.18.5.1';//Master Devices NetID 
	tSync                               : TIME   :=T#3S;                       //interval of Ehercat Managment time
	iMoveStep                           : UINT   :=0; 
	TON_Sync                            : TON ;
	i                                   : USINT  :=0;
    TRIG_Reset                          : R_TRIG;
	iResetCounter                       : SINT  :=-27;                          //1.set state counter  2.startup OP maxtime = 3-(27)*tSync =90s
	(**************************Funtion: Get Master variables**************************)
	fbGetMasterState                    : FB_EcGetMasterState;	
	wCurrentMasterState                 : WORD;                                //master state
	(**************************Funtion: Get Slave Address**************************)
	fbGetAllSlaveAddr                   : FB_EcGetAllSlaveAddr;
    arrBoxAddr                          : ARRAY[0..6] OF UINT;	              //slave address
	(**************************Funtion: Get Slave variables**************************)
	fbGetAllSlaveStates                 : FB_EcGetAllSlaveStates; 
	arrCurrentSlaveState                : ARRAY[0..6] OF ST_EcSlaveState;     //all slaves state	
	(**************************Funtion: Contrl Master State **************************)
	fbSetMasterState                    : FB_EcSetMasterState;
	(**************************Funtion: Contrl Slave State **************************)
	fbSetSlaveState                     : FB_EcSetSlaveState;
	


END_VAR




TRIG_Reset(CLK:=bResetState);
IF TRIG_Reset.Q  THEN
   iResetCounter :=0;	
END_IF

bResetBusy := iResetCounter <=2;
 
CASE iMoveStep OF 
	(*************interval sync of Ehercat Manage***************)
	0:		
	    TON_Sync(IN:=TRUE , PT:=tSync);
		IF TON_Sync.Q   THEN
		   TON_Sync(IN:=FALSE);
		   MasterNetId:=GetMasterNetId(arrAMSNETID:=arrbyNetId);//convert AMSNETID(linked) to T_AmsNetID(fbInput)
		   iMoveStep:=100;
		END_IF
		
	(*************get master state***************)	
	100:
	    fbGetMasterState(sNetId:=MasterNetId, bExecute:=TRUE);		
		iMoveStep:=150;
	150:
	    fbGetMasterState(bExecute:=FALSE);
		IF NOT fbGetMasterState.bBusy  THEN
			   wCurrentMasterState := fbGetMasterState.state;
			   iMoveStep    :=200;
		END_IF
	
    (*************get slaves boxID***************)				
	200:
	    fbGetAllSlaveAddr(sNetId:=MasterNetId, pAddrBuf := ADR(arrBoxAddr), cbBufLen:= SIZEOF(arrBoxAddr),bExecute:=TRUE);
		iMoveStep:=250;
	250:
	    fbGetAllSlaveAddr(bExecute:=FALSE);
		IF NOT fbGetAllSlaveAddr.bBusy  THEN
			   iMoveStep    :=300;
		END_IF
	
    (*************use boxID to get slaves state and buslink***************)		
	300:
	    fbGetAllSlaveStates(sNetId:=MasterNetId, pStateBuf := ADR(arrCurrentSlaveState), cbBufLen:=SIZEOF(arrCurrentSlaveState), bExecute:=TRUE);
		iMoveStep:=350;
	350:
	    fbGetAllSlaveStates(bExecute:=FALSE);	
	    IF NOT fbGetAllSlaveStates.bBusy  THEN
			   iSlavesCount :=fbGetAllSlaveStates.nSlaves;
			   iMoveStep    :=400;
		END_IF
		
    (*************all State to RTC***************)	
    400:
		wAllState.0 := wCurrentMasterState=EC_DEVICE_STATE_OP;
		wAllState.1 := arrCurrentSlaveState[0].deviceState=EC_DEVICE_STATE_OP;
		wAllState.2 := arrCurrentSlaveState[1].deviceState=EC_DEVICE_STATE_OP;
		wAllState.3 := arrCurrentSlaveState[2].deviceState=EC_DEVICE_STATE_OP;
		wAllState.4 := arrCurrentSlaveState[3].deviceState=EC_DEVICE_STATE_OP;
		wAllState.5 := arrCurrentSlaveState[4].deviceState=EC_DEVICE_STATE_OP;
		wAllState.6 := arrCurrentSlaveState[5].deviceState=EC_DEVICE_STATE_OP;
		wAllState.7 := arrCurrentSlaveState[6].deviceState=EC_DEVICE_STATE_OP;
		iMoveStep   := 450;
		
    (*************condition of reset master and slave to OP***************)	
	450://set all bus node to OP 3 times 
	    IF iResetCounter <=2   THEN
		   iResetCounter :=iResetCounter+1;
		   iMoveStep     :=500;
		ELSE  
           iMoveStep     :=0;		  
		END_IF
		
    (*************set master state in OP***************)			
	500:
        IF wCurrentMasterState <> EC_DEVICE_STATE_OP   THEN 	
	       fbSetMasterState(sNetId:=MasterNetId, bExecute:=TRUE, reqState:=EC_DEVICE_STATE_OP);
		END_IF    
		iMoveStep:=550;
	550:
	    fbSetMasterState(bExecute:=FALSE);
		IF NOT fbSetMasterState.bBusy  THEN
			   iMoveStep:=600;
		END_IF
	
	(*************set all slave state follow master state***************)
	600:
	    IF arrBoxAddr[i]>0 AND arrCurrentSlaveState[i].deviceState <> wCurrentMasterState THEN
	       fbSetSlaveState(sNetId:=MasterNetId , nSlaveAddr:=arrBoxAddr[i], bExecute:=TRUE , reqState:=wCurrentMasterState);
		END_IF
		iMoveStep:=650;	
	650://trigger 7 times of iMoveStep=600 to check all slaves in arry
	    fbSetSlaveState(bExecute:=FALSE);
		IF NOT fbSetSlaveState.bBusy  THEN			
			IF     i < 6    THEN
				   i          :=i+1;
				   iMoveStep  :=600;
			ELSE 
  		           i          :=0;
			       iMoveStep  :=0;
			END_IF				 
		END_IF	

END_CASE;

METHOD GetMasterNetId : T_AmsNetID   //convert AMSNETID to T_AMSNETID
VAR_INPUT
	arrAMSNETID     : AMSNETID; 
END_VAR
VAR
	str23Temp       : STRING;
	strSymbol       : STRING:='.';
END_VAR

str23Temp     := CONCAT(STR1:=BYTE_TO_STRING(arrbyNetId[0]) , STR2:=strSymbol);
str23Temp     := CONCAT(STR1:=str23Temp , STR2:=BYTE_TO_STRING(arrbyNetId[1]));
str23Temp     := CONCAT(STR1:=str23Temp , STR2:=strSymbol);
str23Temp     := CONCAT(STR1:=str23Temp , STR2:=BYTE_TO_STRING(arrbyNetId[2]));
str23Temp     := CONCAT(STR1:=str23Temp , STR2:=strSymbol);
str23Temp     := CONCAT(STR1:=str23Temp , STR2:=BYTE_TO_STRING(arrbyNetId[3]));
str23Temp     := CONCAT(STR1:=str23Temp , STR2:=strSymbol);
str23Temp     := CONCAT(STR1:=str23Temp , STR2:=BYTE_TO_STRING(arrbyNetId[4]));
str23Temp     := CONCAT(STR1:=str23Temp , STR2:=strSymbol);
str23Temp     := CONCAT(STR1:=str23Temp , STR2:=BYTE_TO_STRING(arrbyNetId[5]));
str23Temp  	  := CONCAT(STR1:=str23Temp , STR2:=strSymbol);
GetMasterNetId:= str23Temp;
END_METHOD

END_PROGRAM

// ---- POUs/bsm.TcPOU
PROGRAM bsm
VAR
//	bsm_bControlModeHMI	:BOOL	:=FALSE;	//true = use HMI control, false = use etherCAT control

	bsm_intAICollP1 AT %I*	:INT;	//EL3004 #1 CH1, +/-10V -> -32767 to 32768
	bsm_fCollP1	AT %Q*:REAL;
	bsm_intAICollP2 AT %I*	:INT;	//EL3004 #1 CH2, +/-10V -> -32767 to 32768
	bsm_fCollP2	AT %Q*:REAL;
	bsm_intAIJaw1P1 AT %I*	:INT;	//EL3004 #1 CH3, +/-10V -> -32767 to 32768
	bsm_fJaw1P1	AT %Q*:REAL;
	bsm_intAIJaw1P2 AT %I*	:INT;	//EL3004 #1 CH4, +/-10V -> -32767 to 32768
	bsm_fJaw1P2	AT %Q*:REAL;

	bsm_intAIJaw2P1 AT %I*	:INT;	//EL3004 #2 CH1, +/-10V -> -32767 to 32768
	bsm_fJaw2P1	AT %Q*:REAL;
	bsm_intAIJaw2P2 AT %I*	:INT;	//EL3004 #2 CH2, +/-10V -> -32767 to 32768
	bsm_fJaw2P2	AT %Q*:REAL;
	bsm_intAIJaw3P1 AT %I*	:INT;	//EL3004 #2 CH3, +/-10V -> -32767 to 32768
	bsm_fJaw3P1	AT %Q*:REAL;
	bsm_intAIJaw3P2 AT %I*	:INT;	//EL3004 #2 CH4, +/-10V -> -32767 to 32768
	bsm_fJaw3P2	AT %Q*:REAL;
	
	bsm_intAIJaw4P1 AT %I*	:INT;	//EL3004 #3 CH1, +/-10V -> -32767 to 32768
	bsm_fJaw4P1	AT %Q*:REAL;
	bsm_intAIJaw4P2 AT %I*	:INT;	//EL3004 #3 CH2, +/-10V -> -32767 to 32768
	bsm_fJaw4P2	AT %Q*:REAL;
	
	bsm_intAOCollSet AT %Q*	:INT;	//EL4034 #1 CH1, -32767 to 32768 -> +/-10V
//	bsm_fCollSet	:REAL;
	bsm_ethercat_fCollSet	AT %I*:REAL;
	bsm_intAOLwJ4Set AT %Q*	:INT;	//EL4034 #1 CH2, -32767 to 32768 -> +/-10V
//	bsm_fLowJaw4Set	:REAL;
	bsm_ethercat_fLowJaw4Set	AT %I*:REAL;
	bsm_intAOLwJ3Set AT %Q*	:INT;	//EL4034 #1 CH3, -32767 to 32768 -> +/-10V
//	bsm_fLowJaw3Set	:REAL;
	bsm_ethercat_fLowJaw3Set	AT %I*:REAL;
	
	bsm_intAOUpJ2Set AT %Q*	:INT;	//EL4034 #2 CH1, -32767 to 32768 -> +/-10V
//	bsm_fUpJaw2Set	:REAL;
	bsm_ethercat_fUpJaw2Set	AT %I*:REAL;
	bsm_intAOUpJ1Set AT %Q*	:INT;	//EL4034 #2 CH2, -32767 to 32768 -> +/-10V
//	bsm_fUpJaw1Set	:REAL;
	bsm_ethercat_fUpJaw1Set	AT %I*:REAL;
	
	bsm_bFieldLight AT %Q*	:BOOL	:=FALSE;	//EL2008 CH1
	bsm_bRangeFinder AT %Q*	:BOOL	:=FALSE;	//EL2008 CH2
	bsm_bJawBreaker AT %Q*	:BOOL	:=FALSE;	//EL2008 CH3
	bsm_bBSMOK AT %Q*	:BOOL	:=FALSE;	//EL2008 CH4
	bsm_ethercat_bFieldLight AT %I*	:BOOL;
	bsm_ethercat_bRangeFinder AT %I*	:BOOL;
	bsm_ethercat_bJawBreaker AT %I*	:BOOL;
	bsm_ethercat_bBSMOK AT %I*	:BOOL;
END_VAR

//Convert AI int to +/- 10V

bsm_fCollP1:=F_scale_int_real(bsm_intAICollP1);
bsm_fCollP2:=F_scale_int_real(bsm_intAICollP2);

bsm_fJaw1P1:=F_scale_int_real(bsm_intAIJaw1P1);
bsm_fJaw1P2:=F_scale_int_real(bsm_intAIJaw1P2);

bsm_fJaw2P1:=F_scale_int_real(bsm_intAIJaw2P1);
bsm_fJaw2P2:=F_scale_int_real(bsm_intAIJaw2P2);

bsm_fJaw3P1:=F_scale_int_real(bsm_intAIJaw3P1);
bsm_fJaw3P2:=F_scale_int_real(bsm_intAIJaw3P2);

bsm_fJaw4P1:=F_scale_int_real(bsm_intAIJaw4P1);
bsm_fJaw4P2:=F_scale_int_real(bsm_intAIJaw4P2);

//IF NOT bsm_bControlModeHMI THEN
//	bsm_fCollSet := bsm_ethercat_fCollSet;
//	bsm_fLowJaw4Set := bsm_ethercat_fLowJaw4Set;
//	bsm_fLowJaw3Set := bsm_ethercat_fLowJaw3Set;
//	bsm_fUpJaw2Set := bsm_ethercat_fUpJaw2Set;
//	bsm_fUpJaw1Set := bsm_ethercat_fUpJaw1Set;
	bsm_bFieldLight := bsm_ethercat_bFieldLight;
	bsm_bRangeFinder := bsm_ethercat_bRangeFinder;
	bsm_bJawBreaker := bsm_ethercat_bJawBreaker;
	bsm_bBSMOK := bsm_ethercat_bBSMOK;
//END_IF

bsm_intAOCollSet :=F_scale_real_int(bsm_ethercat_fCollSet);
bsm_intAOLwJ4Set :=F_scale_real_int(bsm_ethercat_fLowJaw4Set);
bsm_intAOLwJ3Set :=F_scale_real_int(bsm_ethercat_fLowJaw3Set);
bsm_intAOUpJ2Set :=F_scale_real_int(bsm_ethercat_fUpJaw2Set);
bsm_intAOUpJ1Set :=F_scale_real_int(bsm_ethercat_fUpJaw1Set);

END_PROGRAM

// ---- POUs/F_scale_int_real.TcPOU
FUNCTION F_scale_int_real : real
VAR_INPUT
	intput_int	:INT;
END_VAR
VAR
	scaled_real	:REAL;
END_VAR

//Sacle INT to +/-10V
IF (intput_int>=0) THEN
	scaled_real := INT_TO_REAL(ABS(intput_int))*10/32767;
ELSE
	scaled_real := - INT_TO_REAL(ABS(intput_int))*10/32767;
END_IF

F_scale_int_real:=LIMIT(-10,scaled_real,10);

END_FUNCTION

// ---- POUs/F_scale_real_int.TcPOU
FUNCTION F_scale_real_int : INT
VAR_INPUT
	input_real	:REAL;
END_VAR
VAR
	scaled_int	:int;
END_VAR

//Sacle +/-10V to INT
input_real:=LIMIT(-10,input_real,10);

IF (input_real>=0) THEN
	scaled_int := REAL_TO_INT(ABS(input_real)/10*32767);
ELSE
	scaled_int := - REAL_TO_INT(ABS(input_real)/10*32767);
END_IF

F_scale_real_int:=LIMIT(-32767,scaled_int,32767);

END_FUNCTION

// ---- POUs/BeamEnChain.TcPOU
PROGRAM BeamEnChain
VAR
	BeamEn	AT %Q*:BOOL;
END_VAR

BeamEn := TRUE;

END_PROGRAM

// ---- POUs/OnGantry_IO.TcPOU
PROGRAM OnGantry_IO
VAR
	//watchdog
	intBoneCounter	:INT	:=0;
	tonSwReset :TON;
	tpSwReset :Tp;
	
	//Interface of IO To RTC		
	plc_to_io_bGantryTouchGuard   AT%I*   : BOOL;
	plc_to_cpp_bGantryTouchGuard  AT%Q*   : BOOL;
	
	plc_to_io_bAutoMove           AT%I*   : BOOL;
	plc_to_cpp_bAutoMove          AT%Q*   : BOOL;
	
	plc_to_io_OnGantryRtcWdOK     AT%I*   : BOOL;
	plc_to_cpp_OnGantryRtcWdOK    AT%Q*   : BOOL;
	
	plc_to_io_bCanOpenOk          AT%Q*   : BOOL;
	plc_to_cpp_bCanOpenOk         AT%I*   : BOOL;
		
	plc_to_io_OnGantryMoveEn      AT%Q*   : BOOL;
	plc_to_cpp_OnGantryMoveEn     AT%I*   : BOOL;
		
	plc_to_io_bSwWatchDogService  AT%Q*   : BOOL;
	
	plc_to_io_bSwRest             AT%Q*   : BOOL;
	plc_to_cpp_bSwRest            AT%I*   : BOOL;
	
	plc_to_io_bKvEn               AT%Q*   : BOOL;
	plc_to_cpp_bKvEn              AT%I*   : BOOL;
	
	plc_to_io_bEthercatInOk       AT%Q*   : BOOL;
	plc_to_cpp_bEthercatInOk      AT%I*   : BOOL;
	
	plc_to_io_bEthercatOutOk      AT%Q*   : BOOL;
	plc_to_cpp_bEthercatOutOk     AT%I*   : BOOL;	
	
	plc_to_cpp_bSwManualMotionEn  AT%I*		:BOOL;
	plc_to_io_bSwManualMotionEn   AT%Q*		:BOOL;
END_VAR

IF intBoneCounter >= 4 THEN
	plc_to_io_bSwWatchDogService := NOT plc_to_io_bSwWatchDogService;		//Flip bone to feed the dog
	intBoneCounter := 0;
ELSE intBoneCounter := intBoneCounter + 1; 
END_IF

IF plc_to_io_bSwRest AND (NOT plc_to_cpp_bSwRest) THEN		// turn io signal to false in next cycle if cpp signal is false
	plc_to_io_bSwRest := FALSE;
END_IF

tpSwReset(IN:=TwinCAT_SystemInfoVarList._TaskInfo[Tc2_System.GETCURTASKINDEXEX()].FirstCycle,PT:=T#2S,Q=>,ET=>);
tonSwReset(IN:=tpSwReset.Q,PT:=T#1S,Q=>,ET=>);		//Reset pulse will send after 1sec of PLC first cycle

plc_to_io_bSwRest := plc_to_cpp_bSwRest OR tonSwReset.Q;

io_update();

ACTION io_update:


////****beta interface of plc and cpp****////
//inputIO to plc to cpp	
plc_to_cpp_bGantryTouchGuard := plc_to_io_bGantryTouchGuard;
plc_to_cpp_bAutoMove := plc_to_io_bAutoMove;        
plc_to_cpp_OnGantryRtcWdOK  := plc_to_io_OnGantryRtcWdOK ;
     
     
plc_to_io_bCanOpenOk :=	plc_to_cpp_bCanOpenOk;
plc_to_io_OnGantryMoveEn := plc_to_cpp_OnGantryMoveEn;    	
plc_to_io_bSwRest := plc_to_cpp_bSwRest;          	         	
plc_to_io_bKvEn :=  plc_to_cpp_bKvEn;        
plc_to_io_bEthercatOutOk := plc_to_cpp_bEthercatOutOk;
plc_to_io_bEthercatInOk := plc_to_cpp_bEthercatInOk; 

plc_to_io_bSwManualMotionEn:=plc_to_cpp_bSwManualMotionEn;
END_ACTION

END_PROGRAM
